TYPE ST_PV_data :
STRUCT
	Line_current_L1		:DINT;
	Line_current_L2		:DINT;
	Line_current_L3		:DINT;
	PV_Power			:DWORD;
END_STRUCT
END_TYPE

(* stored: Version 1.1.0.1, ProductVersion 3.1.4020.6
   DUT ST_PV_data: Id {8a885483-9610-44f8-ae2a-6d919aab885e} *)
